FUNCTION_BLOCK FB_ParallelJobContainerCreator IMPLEMENTS InterfaceTaskCreator
VAR_INPUT
END_VAR
VAR_OUTPUT
END_VAR
VAR
END_VAR

{warning 'add method implementation '}
METHOD create_future : InterfaceFuture
VAR_INPUT
	future_name	: STRING;
END_VAR
VAR
	_p_future : POINTER TO FB_ParallelJobContainer;
END_VAR
_p_future := __NEW(FB_ParallelJobContainer);
_p_future^.future_name := future_name;
create_future := _p_future^;
END_METHOD

{warning 'add method implementation '}
METHOD destroy_future : InterfaceFuture
VAR_INPUT
	future	: InterfaceFuture;
END_VAR
VAR
	_p_future : POINTER TO FB_ParallelJobContainer;
END_VAR
IF __QUERYPOINTER(future, _p_future) THEN
	__DELETE(_p_future);
	IF _p_future = 0  THEN
		destroy_future := 0;
	END_IF
END_IF
END_METHOD

END_FUNCTION_BLOCK

(* stored: Version 1.1.0.1, ProductVersion 3.1.4026.13
   POU FB_ParallelJobContainerCreator: Id {808db55b-c727-45ae-8e1f-ebf797e858e3}, SpecialFunc None
   Method create_future: Id {f7e25f65-449b-4ef3-a719-946b3d87fba9}
   Method destroy_future: Id {059ba90e-ca78-49a7-9d25-013656fe00e0} *)
